FUNCTION_BLOCK FB_F_TRIG (* Detect falling edge *)
  (* Standard: 61499-1; Description: Copyright (c) 2023 Martin Erich Jobst This program and the accompanying materials are made available under the terms of the Eclipse Public License 2.0 which is available at https://www.eclipse.org/legal/epl-2.0/ SPDX-License-Identifier: EPL-2.0 *)
  (* Version 1.0, 2023-04-28, Martin Jobst *)
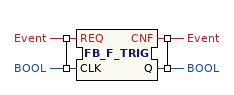
  EVENT_INPUT
    REQ WITH CLK; (* Normal Execution Request *)
  END_EVENT
  EVENT_OUTPUT
    CNF WITH Q; (* Execution Confirmation *)
  END_EVENT
  VAR_INPUT
    CLK : BOOL; (* Clock *)
  END_VAR
  VAR_OUTPUT
    Q : BOOL; (* Output *)
  END_VAR
  VAR
    MEM : BOOL := TRUE;
  END_VAR
  ALGORITHM REQ IN ST:
Q := NOT CLK AND NOT MEM;
MEM := NOT CLK;
  END_ALGORITHM
END_FUNCTION_BLOCK
